FUNCTION_BLOCK Selector (* Basic Function Block Type *)
  (* Standard: 61499-2 *)
  (* Version 0.0, 2011-12-23, 4DIAC-IDE, 4DIAC-Consortium *)
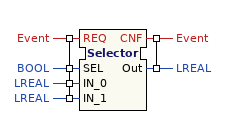
  EVENT_INPUT
    REQ WITH SEL, IN_0, IN_1; (* Normal Execution Request *)
  END_EVENT
  EVENT_OUTPUT
    CNF WITH Out; (* Execution Confirmation *)
  END_EVENT
  VAR_INPUT
    SEL : BOOL; (* Input event qualifier *)
    IN_0 : LREAL;
    IN_1 : LREAL;
  END_VAR
  VAR_OUTPUT
    Out : LREAL; (* Output event qualifier *)
  END_VAR
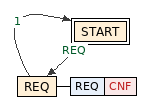
  EC_STATES
    START; (* Initial State *)
    REQ : REQ -> CNF; (* Normal execution *)
  END_STATES
  EC_TRANSITIONS
    START TO REQ := REQ;
    REQ TO START := 1;
  END_TRANSITIONS
  ALGORITHM REQ IN ST: (* Normally executed algorithm *)
IF SEL = 1 THEN
	Out := IN_1;
ELSE
	Out:= IN_0;
END_IF;
  END_ALGORITHM
END_FUNCTION_BLOCK
